// LS Electric XG5000 project: test
// PLC LSPLC

PROGRAM NewProgram (task: 스캔 프로그램)

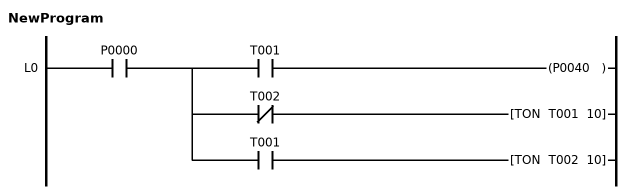
; L0
LOAD      P0000
MPUSH
AND       T001
OUT       P0040
MLOAD
AND NOT   T002
TON       T001 10
MPOP
AND       T001
TON       T002 10